// TIA Portal V21 export
TYPE "Campionatura"
   STRUCT
      OrarioCampionatura : Date_And_Time;
      MetriCubi : Real;
   END_STRUCT;
END_TYPE
